(* IEC 61131-3 sources: Structured-Text/Source Code/Utility/DIDOREF, 2 files *)

(* ---- DIDOREF.ST ---- *)
IF Invert THEN
	Output := NOT Input;
	Inverted := True;
ELSE
	Output := Input;
	Inverted := False;
END_IF;

(* ---- Local Variables.ST ---- *)
VAR_INPUT
	Input:	BOOL;		//Tagname of the Input
END_VAR

VAR_OUTPUT
	Output:		BOOL;	//Output Value
	Inverted:	BOOL;	//Output invert status
END_VAR

VAR
	Invert:	BOOL;
END_VAR
